PROGRAM MAIN
VAR
	_LampIsOn		: BOOL := FALSE;
	_ButtonIsPushed	: BOOL := FALSE;
END_VAR

// This program operates a lamp. When a button is pushed, and held down, the lamp turns on.
// When the button is released, the lamp turns off. Instead of using a real lamp and a button,
// they are in the visualization.

IF _ButtonIsPushed THEN
	_LampIsOn := TRUE;
ELSE
	_LampIsOn := FALSE;
END_IF

END_PROGRAM

(* stored: Version 1.1.0.1
   POU MAIN: Id {2e6786d1-c064-428e-a199-bdaaa8521a4f}, SpecialFunc None *)
